INTERFACE I_Publisher

METHOD AddSubscriber : BOOL
VAR_INPUT
	ipSubscriber : I_Subscriber;
END_VAR
END_METHOD

METHOD RemoveSubscriber : BOOL
VAR_INPUT
	ipSubscriber : I_Subscriber;
END_VAR
END_METHOD

END_INTERFACE

(* stored: Version 1.1.0.1, ProductVersion 3.1.4022.18
   Itf I_Publisher: Id {f50d4c11-a399-4ef5-8b2a-7ec13cf25048}
   Method AddSubscriber: Id {ab6add66-a4a2-4400-ad3b-e6a24cb0baa0}
   Method RemoveSubscriber: Id {18773c0d-16da-4d52-8661-85c823230dc4} *)
